{attribute 'qualified_only'}
TYPE E_State :
(
	Init := 0,
	ReadOnce,
	ReadPeriodically,
	Error,
	
	Idle,
	ReadOnce_CpuUsage,
	ReadOnce_CpuTemperature,
	ReadOnce_SrnMainboard,
	ReadOnce_SrnIPC,
	Write_DHCP,
	Write_IPAddr
	
);
END_TYPE

(* stored: Version 1.1.0.1, ProductVersion 3.1.4024.11
   DUT E_State: Id {152610e0-cdbf-4e25-93df-dac94cd9b39b} *)
